// TIA Portal V15.1 export
// export: Created 2024-06-21T08:41:01.7297827Z, ExportSetting WithDefaults, DisplayName Totally Integrated Automation Portal, DisplayVersion V15.1 Update 5, DisplayName TIA Portal Openness, DisplayVersion V15.1 Update 5, DisplayName SINAMICS Startdrive Advanced, DisplayVersion V15.1, DisplayName G130, G150, S120, S150, SINAMICS MV, S210, DisplayVersion V15.1, DisplayName G110M, G120, G120C, G120D, G120P, DisplayVersion V15.1, DisplayName STEP 7 Professional, DisplayVersion V15.1 Update 5, DisplayName STEP 7 Safety, DisplayVersion V15.1, DisplayName WinCC Professional, DisplayVersion V15.1 Update 5, DisplayName SIMATIC Visualization Architect, DisplayVersion V15.1
FUNCTION_BLOCK "LCounter1Week"   // FB1801, FBD
TITLE = LCounter1Week
{ S7_Optimized_Access := 'FALSE' }
AUTHOR : VCC
FAMILY : Supervis
NAME : LCpt1W
VERSION : 1.0
// ==============================================================================
// Module create to count body produced during all shifts of the week.
// One counter per shift (moring - evening & night) per day (from monday to sunday)
// all total are foreseen.
// 
// --------------------------------------------------------------------
// Day          ! Morning shift ! Evening shift ! Night shift ! total !
// -------------!---------------!---------------!-------------!-------!
// Monday (1)   !               !               !             !       !
// -------------!---------------!---------------!-------------!-------!
// Tuesday (2)  !               !               !             !       !
// -------------!---------------!---------------!-------------!-------!
// Wednesday (3)!               !               !             !       !
// -------------!---------------!---------------!-------------!-------!
// Thursday (4) !               !               !             !       !
// -------------!---------------!---------------!-------------!-------!
// Friday (5)   !               !               !             !       !
// -------------!---------------!---------------!-------------!-------!
// Saturday (6) !               !               !             !       !
// -------------!---------------!---------------!-------------!-------!
// Sunday (7)   !               !               !             !       !
// ====================================================================
// Amount       !               !               !             !       !
// ====================================================================
// Tatal        !=============================================!       !
// ====================================================================
// 
// ==============================================================================
// stored: AutoNumber false, IsIECCheckEnabled false, SetENOAutomatically False, UDAEnableTagReadback false
   VAR_INPUT
      I_CountedInput { ExternalAccessible := 'False'; ExternalVisible := 'False'; ExternalWritable := 'False'} : Bool;   // Value to be counted
      I_MorningShift { ExternalAccessible := 'False'; ExternalVisible := 'False'; ExternalWritable := 'False'} : Bool;   // Morning shift
      I_EveningShift { ExternalAccessible := 'False'; ExternalVisible := 'False'; ExternalWritable := 'False'} : Bool;   // Evening shift
      I_NightShift { ExternalAccessible := 'False'; ExternalVisible := 'False'; ExternalWritable := 'False'} : Bool;   // NightShift
   END_VAR
   VAR_OUTPUT
      H_IAnim { ExternalAccessible := 'False'; ExternalVisible := 'False'; ExternalWritable := 'False'} : Word;   // HMI Animation of the icon
   END_VAR
   VAR DB_SPECIFIC
      H_Out : Struct   // HMI
         Anim : Word;   // HMI Animation of the object
         MorningDay1Value : Int;   // Total Production value Monday (day 1) - Morning Shift
         EveningDay1Value : Int;   // Total Production value Monday (day 1) - Evening Shift
         NightDay1Value : Int;   // Total Production value Monday (day 1) - Night Shift
         MorningDay2Value : Int;   // Total Production value Tuesday (day 2) - Morning Shift
         EveningDay2Value : Int;   // Total Production value Tuesday (day 2) - Evening Shift
         NightDay2Value : Int;   // Total Production value Tuesday (day 2) - Night Shift
         MorningDay3Value : Int;   // Total Production value Wednesday (day 3) - Morning Shift
         EveningDay3Value : Int;   // Total Production value Wednesday (day 3) - Evening Shift
         NightDay3Value : Int;   // Total Production value Wednesday (day 3) - Night Shift
         MorningDay4Value : Int;   // Total Production value Thursday (day 4) - Morning Shift
         EveningDay4Value : Int;   // Total Production value Thursday (day 4) - Evening Shift
         NightDay4Value : Int;   // Total Production value Thursday (day 4) - Night Shift
         MorningDay5Value : Int;   // Total Production value Friday (day 5) - Morning Shift
         EveningDay5Value : Int;   // Total Production value Friday (day 5) - Evening Shift
         NightDay5Value : Int;   // Total Production value Friday (day 5) - Night Shift
         MorningDay6Value : Int;   // Total Production value Saturday (day 6) - Morning Shift
         EveningDay6Value : Int;   // Total Production value Saturday (day 6) - Evening Shift
         NightDay6Value : Int;   // Total Production value Saturday (day 6) - Night Shift
         MorningDay7Value : Int;   // Production value Sunday (day 7) - Morning Shift
         EveningDay7Value : Int;   // Production value Sunday (day 7) - Evening Shift
         NightDay7Value : Int;   // Production value Sunday (day 7) - Night Shift
         Day1Value : Int;   // Total Production value Monday (day 1)
         Day2Value : Int;   // Total Production value tuesday (day 2)
         Day3Value : Int;   // Total Production value Wednesday (day 3)
         Day4Value : Int;   // Total Production value Thursday (day 4)
         Day5Value : Int;   // Total Production value Friday (day 5)
         Day6Value : Int;   // Total Production value Saturday (day 6)
         Day7Value : Int;   // Total Production value Sunday (day 7)
         TotalMorning : Int;   // Total Production value Morning
         TotalEvening : Int;   // Total Production value Evening
         TotalNight : Int;   // Total Production value Night
         WeekValue : Int;   // Total Production value Week
         TotalValue : DInt;   // Total production value
         DBnr : Int;   // HMI Animation DB number
      END_STRUCT;
      CountedInputPulse { ExternalAccessible := 'False'; ExternalVisible := 'False'; ExternalWritable := 'False'} : Bool;   // Pulse of value to be counted
      CountUp { ExternalAccessible := 'False'; ExternalVisible := 'False'; ExternalWritable := 'False'} : Bool;   // Pulse of value to be counted
      MorningShiftPulse { ExternalAccessible := 'False'; ExternalVisible := 'False'; ExternalWritable := 'False'} : Bool;   // Pulse of Morning shift
      MorningPulse { ExternalAccessible := 'False'; ExternalVisible := 'False'; ExternalWritable := 'False'} : Bool;   // Pulse of Morning shift
      Day1 { ExternalAccessible := 'False'; ExternalVisible := 'False'; ExternalWritable := 'False'} : Bool;   // Day 1 = Monday
      Day2 { ExternalAccessible := 'False'; ExternalVisible := 'False'; ExternalWritable := 'False'} : Bool;   // Day 2 = Tuesday
      Day3 { ExternalAccessible := 'False'; ExternalVisible := 'False'; ExternalWritable := 'False'} : Bool;   // Day 3 = Wednesday
      Day4 { ExternalAccessible := 'False'; ExternalVisible := 'False'; ExternalWritable := 'False'} : Bool;   // Day 4 = Thursday
      Day5 { ExternalAccessible := 'False'; ExternalVisible := 'False'; ExternalWritable := 'False'} : Bool;   // Day 5 = Friday
      Day6 { ExternalAccessible := 'False'; ExternalVisible := 'False'; ExternalWritable := 'False'} : Bool;   // Day 6 = Saturday
      Day7 { ExternalAccessible := 'False'; ExternalVisible := 'False'; ExternalWritable := 'False'} : Bool;   // Day 7 = Sunday
      MorningValue { ExternalAccessible := 'False'; ExternalVisible := 'False'; ExternalWritable := 'False'} : Int;   // Morning production value
      EveningValue { ExternalAccessible := 'False'; ExternalVisible := 'False'; ExternalWritable := 'False'} : Int;   // Evening production value
      NightValue { ExternalAccessible := 'False'; ExternalVisible := 'False'; ExternalWritable := 'False'} : Int;   // Night production value
      MorningDay1Value { ExternalAccessible := 'False'; ExternalVisible := 'False'; ExternalWritable := 'False'} : Int;   // Total Production value Monday (day 1) - Morning Shift
      EveningDay1Value { ExternalAccessible := 'False'; ExternalVisible := 'False'; ExternalWritable := 'False'} : Int;   // Total Production value Monday (day 1) - Evening Shift
      NightDay1Value { ExternalAccessible := 'False'; ExternalVisible := 'False'; ExternalWritable := 'False'} : Int;   // Total Production value Monday (day 1) - Night Shift
      MorningDay2Value { ExternalAccessible := 'False'; ExternalVisible := 'False'; ExternalWritable := 'False'} : Int;   // Total Production value Tuesday (day 2) - Morning Shift
      EveningDay2Value { ExternalAccessible := 'False'; ExternalVisible := 'False'; ExternalWritable := 'False'} : Int;   // Total Production value Tuesday (day 2) - Evening Shift
      NightDay2Value { ExternalAccessible := 'False'; ExternalVisible := 'False'; ExternalWritable := 'False'} : Int;   // Total Production value Tuesday (day 2) - Night Shift
      MorningDay3Value { ExternalAccessible := 'False'; ExternalVisible := 'False'; ExternalWritable := 'False'} : Int;   // Total Production value Wednesday (day 3) - Morning Shift
      EveningDay3Value { ExternalAccessible := 'False'; ExternalVisible := 'False'; ExternalWritable := 'False'} : Int;   // Total Production value Wednesday (day 3) - Evening Shift
      NightDay3Value { ExternalAccessible := 'False'; ExternalVisible := 'False'; ExternalWritable := 'False'} : Int;   // Total Production value Wednesday (day 3) - Night Shift
      MorningDay4Value { ExternalAccessible := 'False'; ExternalVisible := 'False'; ExternalWritable := 'False'} : Int;   // Total Production value Thursday (day 4) - Morning Shift
      EveningDay4Value { ExternalAccessible := 'False'; ExternalVisible := 'False'; ExternalWritable := 'False'} : Int;   // Total Production value Thursday (day 4) - Evening Shift
      NightDay4Value { ExternalAccessible := 'False'; ExternalVisible := 'False'; ExternalWritable := 'False'} : Int;   // Total Production value Thursday (day 4) - Night Shift
      MorningDay5Value { ExternalAccessible := 'False'; ExternalVisible := 'False'; ExternalWritable := 'False'} : Int;   // Total Production value Friday (day 5) - Morning Shift
      EveningDay5Value { ExternalAccessible := 'False'; ExternalVisible := 'False'; ExternalWritable := 'False'} : Int;   // Total Production value Friday (day 5) - Evening Shift
      NightDay5Value { ExternalAccessible := 'False'; ExternalVisible := 'False'; ExternalWritable := 'False'} : Int;   // Total Production value Friday (day 5) - Night Shift
      MorningDay6Value { ExternalAccessible := 'False'; ExternalVisible := 'False'; ExternalWritable := 'False'} : Int;   // Total Production value Saturday (day 6) - Morning Shift
      EveningDay6Value { ExternalAccessible := 'False'; ExternalVisible := 'False'; ExternalWritable := 'False'} : Int;   // Total Production value Saturday (day 6) - Evening Shift
      NightDay6Value { ExternalAccessible := 'False'; ExternalVisible := 'False'; ExternalWritable := 'False'} : Int;   // Total Production value Saturday (day 6) - Night Shift
      MorningDay7Value { ExternalAccessible := 'False'; ExternalVisible := 'False'; ExternalWritable := 'False'} : Int;   // Production value Sunday (day 7) - Morning Shift
      EveningDay7Value { ExternalAccessible := 'False'; ExternalVisible := 'False'; ExternalWritable := 'False'} : Int;   // Production value Sunday (day 7) - Evening Shift
      NightDay7Value { ExternalAccessible := 'False'; ExternalVisible := 'False'; ExternalWritable := 'False'} : Int;   // Production value Sunday (day 7) - Night Shift
      Day1Value { ExternalAccessible := 'False'; ExternalVisible := 'False'; ExternalWritable := 'False'} : Int;   // Total Production value Monday (day 1)
      Day2Value { ExternalAccessible := 'False'; ExternalVisible := 'False'; ExternalWritable := 'False'} : Int;   // Total Production value tuesday (day 2)
      Day3Value { ExternalAccessible := 'False'; ExternalVisible := 'False'; ExternalWritable := 'False'} : Int;   // Total Production value Wednesday (day 3)
      Day4Value { ExternalAccessible := 'False'; ExternalVisible := 'False'; ExternalWritable := 'False'} : Int;   // Total Production value Thursday (day 4)
      Day5Value { ExternalAccessible := 'False'; ExternalVisible := 'False'; ExternalWritable := 'False'} : Int;   // Total Production value Friday (day 5)
      Day6Value { ExternalAccessible := 'False'; ExternalVisible := 'False'; ExternalWritable := 'False'} : Int;   // Total Production value Saturday (day 6)
      Day7Value { ExternalAccessible := 'False'; ExternalVisible := 'False'; ExternalWritable := 'False'} : Int;   // Total Production value Sunday (day 7)
      WeekValue { ExternalAccessible := 'False'; ExternalVisible := 'False'; ExternalWritable := 'False'} : Int;   // Total Production value Week
      TotalValue { ExternalAccessible := 'False'; ExternalVisible := 'False'; ExternalWritable := 'False'} : DInt;   // Total production value
      DBnr { ExternalAccessible := 'False'; ExternalVisible := 'False'; ExternalWritable := 'False'} : Int;   // HMI DB number
   END_VAR
   VAR_TEMP   // added for the SCL form of the ladder/FBD networks
      _w1 : Bool;
   END_VAR
BEGIN

NETWORK
TITLE = **** 1 - Inputs **** DB number
// DB number
      L     DINO;
      T     #DBnr;

REGION Network 2: **** 4.4 - Machine status - Calculated **** Total production counter
   // Total production counter
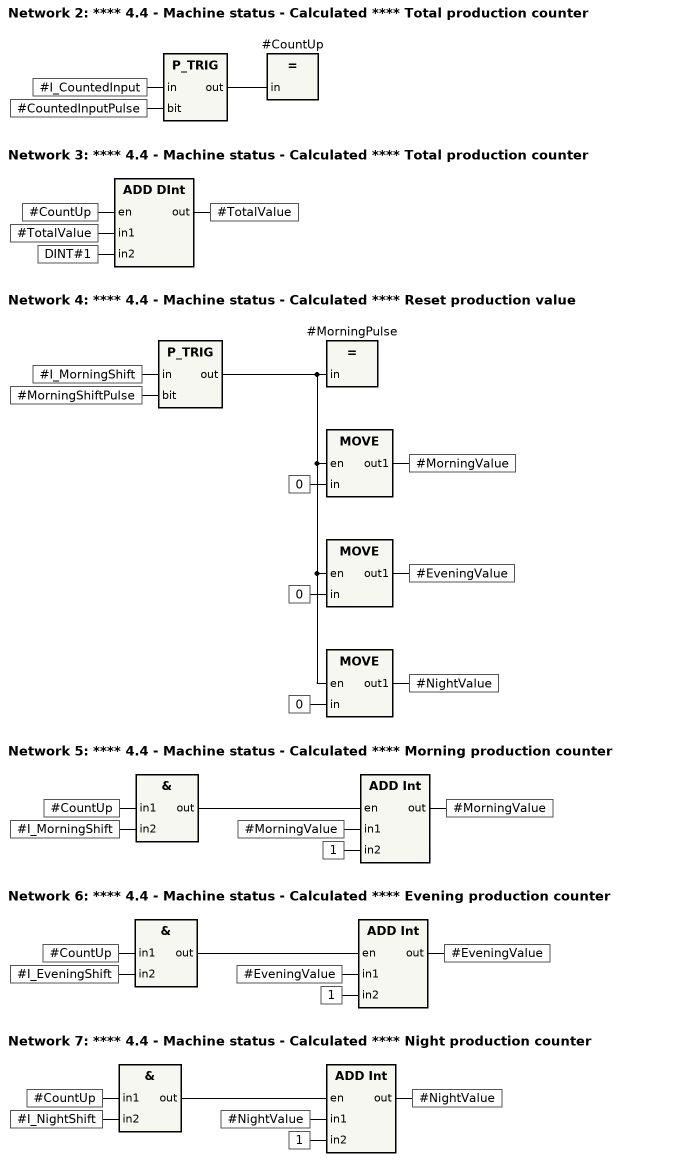
   #_w1 := #I_CountedInput AND NOT #CountedInputPulse;   // rising edge
   #CountedInputPulse := #I_CountedInput;
   #CountUp := #_w1;
END_REGION

REGION Network 3: **** 4.4 - Machine status - Calculated **** Total production counter
   // Total production counter
   IF #CountUp THEN #TotalValue := #TotalValue + DINT#1; END_IF;
END_REGION

REGION Network 4: **** 4.4 - Machine status - Calculated **** Reset production value
   // Reset production value
   #_w1 := #I_MorningShift AND NOT #MorningShiftPulse;   // rising edge
   #MorningShiftPulse := #I_MorningShift;
   #MorningPulse := #_w1;
   IF #_w1 THEN
       #MorningValue := 0;
       #EveningValue := 0;
       #NightValue := 0;
   END_IF;
END_REGION

REGION Network 5: **** 4.4 - Machine status - Calculated **** Morning production counter
   // Morning production counter
   IF #CountUp AND #I_MorningShift THEN #MorningValue := #MorningValue + 1; END_IF;
END_REGION

REGION Network 6: **** 4.4 - Machine status - Calculated **** Evening production counter
   // Evening production counter
   IF #CountUp AND #I_EveningShift THEN #EveningValue := #EveningValue + 1; END_IF;
END_REGION

REGION Network 7: **** 4.4 - Machine status - Calculated **** Night production counter
   // Night production counter
   IF #CountUp AND #I_NightShift THEN #NightValue := #NightValue + 1; END_IF;
END_REGION

REGION Network 8: **** 4.4 - Machine status - Calculated **** Set Monday - reset other days
   // Set Monday - reset other days
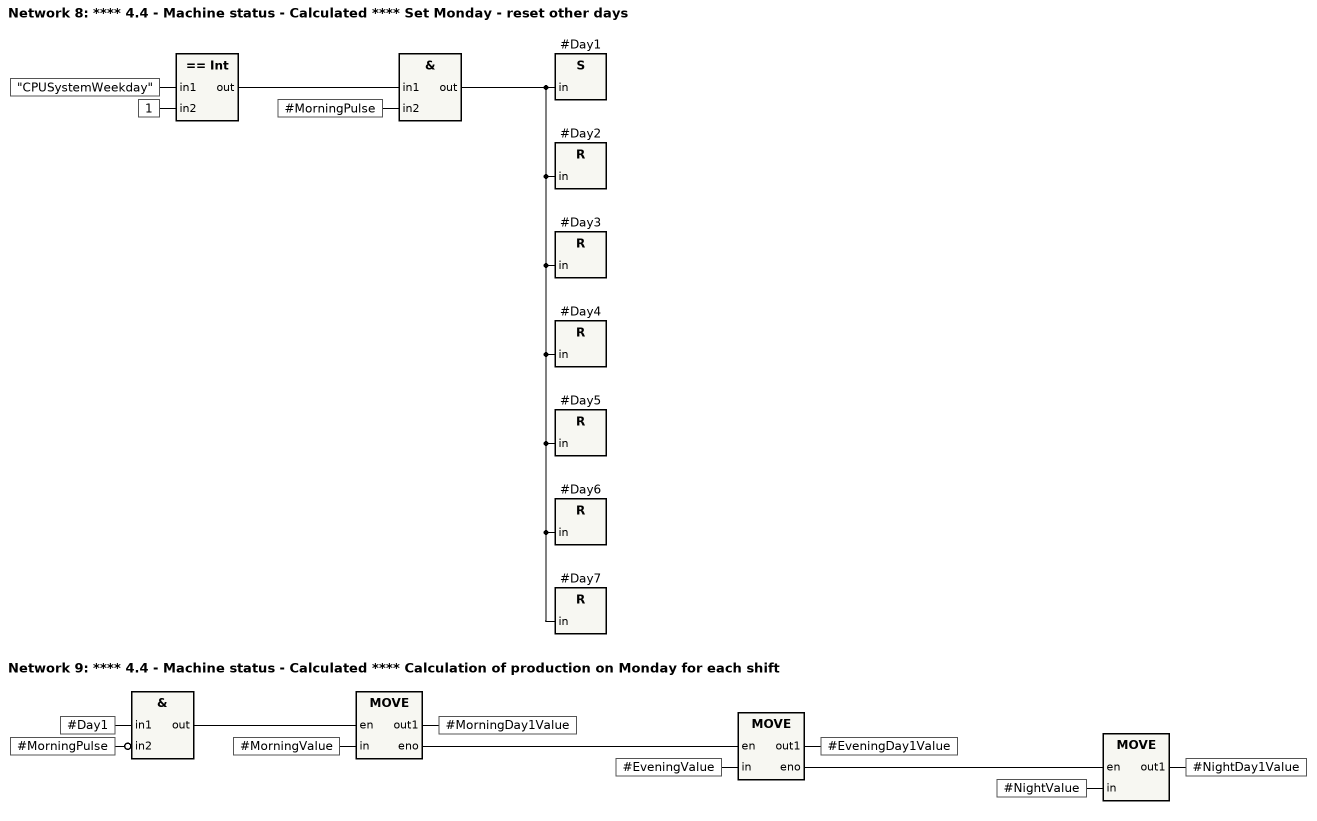
   IF ("CPUSystemWeekday" = 1) AND #MorningPulse THEN
       #Day1 := TRUE;
       #Day2 := FALSE;
       #Day3 := FALSE;
       #Day4 := FALSE;
       #Day5 := FALSE;
       #Day6 := FALSE;
       #Day7 := FALSE;
   END_IF;
END_REGION

REGION Network 9: **** 4.4 - Machine status - Calculated **** Calculation of production on Monday for each shift
   // Calculation of production on Monday for each shift
   // ENO of a box is taken as its EN; it also drops when the box reports an error
   IF #Day1 AND NOT #MorningPulse THEN
       #MorningDay1Value := #MorningValue;
       #EveningDay1Value := #EveningValue;
       #NightDay1Value := #NightValue;
   END_IF;
END_REGION

NETWORK
TITLE = **** 4.4 - Machine status - Calculated **** Total production on Monday
// Total production on Monday
      L     #MorningDay1Value;  // amount of bodies on day 1 - Morning shift (Monday)
      L     #EveningDay1Value;  // amount of bodies on day 1 - Evening shift (Monday)
      +I;
      L     #NightDay1Value;  // amount of bodies on day 1 - Night shift (Monday)
      +I;
      T     #Day1Value;  // amount of bodies on day 1 (Monday)

REGION Network 11: **** 4.4 - Machine status - Calculated **** Set Tuesday - reset other days
   // Set Tuesday - reset other days
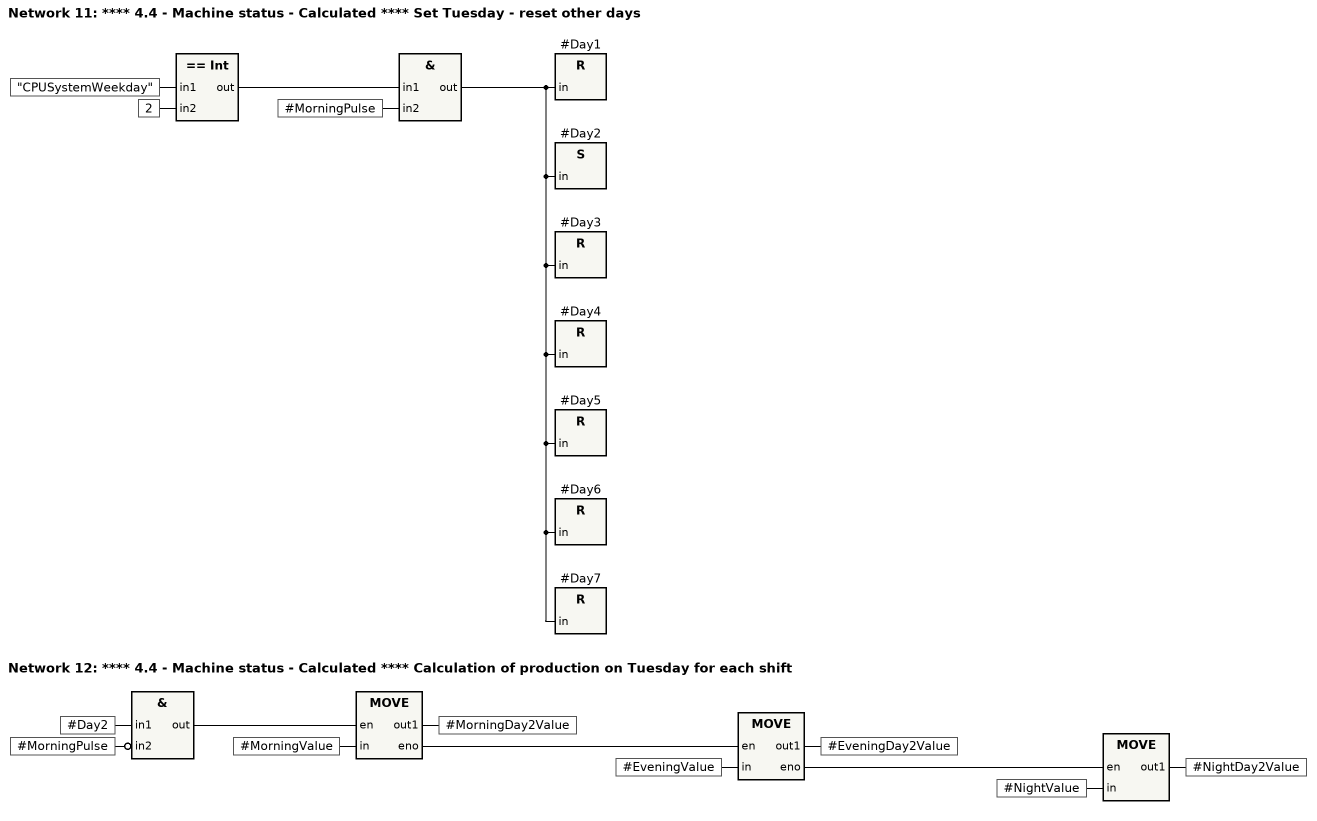
   IF ("CPUSystemWeekday" = 2) AND #MorningPulse THEN
       #Day1 := FALSE;
       #Day2 := TRUE;
       #Day3 := FALSE;
       #Day4 := FALSE;
       #Day5 := FALSE;
       #Day6 := FALSE;
       #Day7 := FALSE;
   END_IF;
END_REGION

REGION Network 12: **** 4.4 - Machine status - Calculated **** Calculation of production on Tuesday for each shift
   // Calculation of production on Tuesday for each shift
   // ENO of a box is taken as its EN; it also drops when the box reports an error
   IF #Day2 AND NOT #MorningPulse THEN
       #MorningDay2Value := #MorningValue;
       #EveningDay2Value := #EveningValue;
       #NightDay2Value := #NightValue;
   END_IF;
END_REGION

NETWORK
TITLE = **** 4.4 - Machine status - Calculated **** Total production on Thuesday
// Total production on Thuesday
      L     #MorningDay2Value;  // amount of bodies on day 2 - Morning shift (Tuesday)
      L     #EveningDay2Value;  // amount of bodies on day 2 - Evening shift (Tuesday)
      +I;
      L     #NightDay2Value;  // amount of bodies on day 2 - Night shift (Tuesday)
      +I;
      T     #Day2Value;  // amount of bodies on day 2 (Tuesday)

REGION Network 14: **** 4.4 - Machine status - Calculated **** Set Wednesday - reset other days
   // Set Wednesday - reset other days
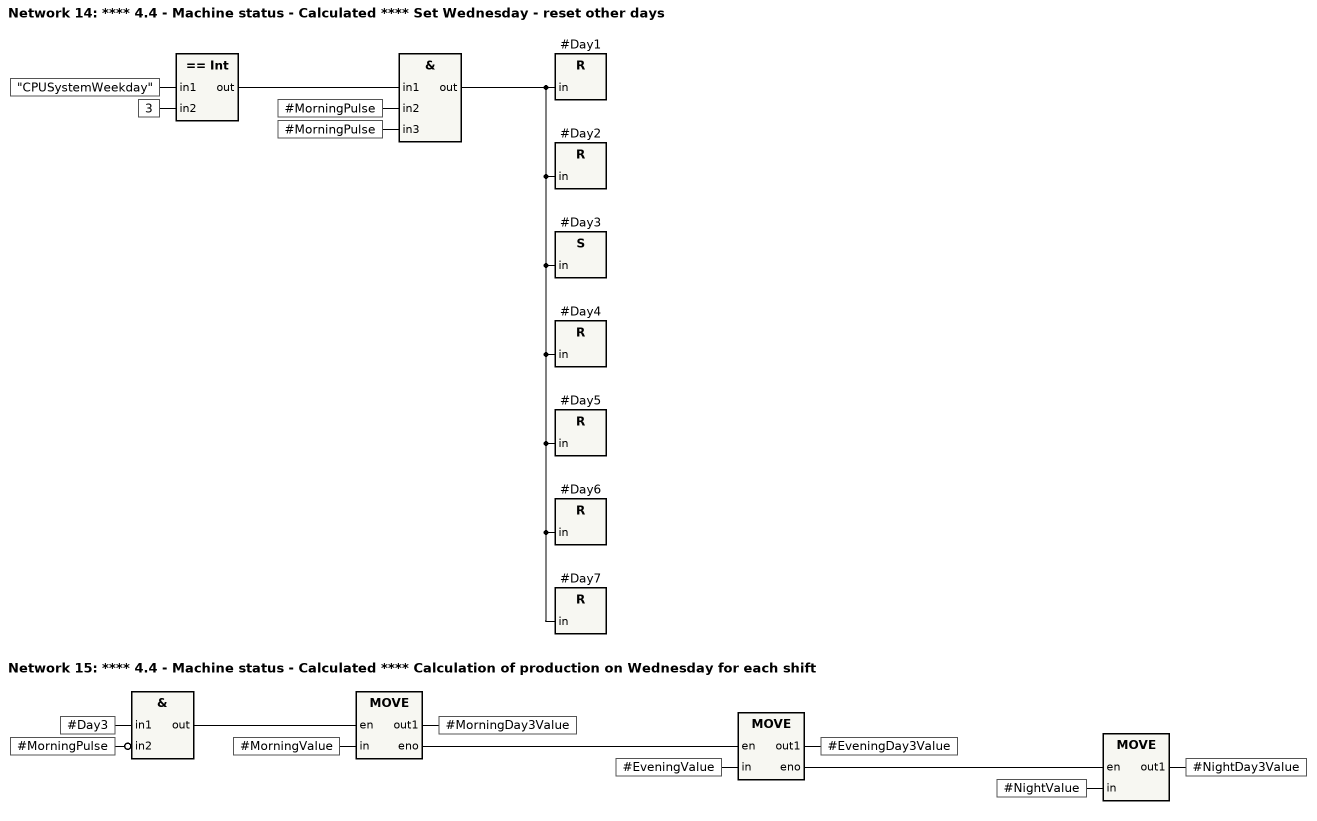
   IF ("CPUSystemWeekday" = 3) AND #MorningPulse AND #MorningPulse THEN
       #Day1 := FALSE;
       #Day2 := FALSE;
       #Day3 := TRUE;
       #Day4 := FALSE;
       #Day5 := FALSE;
       #Day6 := FALSE;
       #Day7 := FALSE;
   END_IF;
END_REGION

REGION Network 15: **** 4.4 - Machine status - Calculated **** Calculation of production on Wednesday for each shift
   // Calculation of production on Wednesday for each shift
   // ENO of a box is taken as its EN; it also drops when the box reports an error
   IF #Day3 AND NOT #MorningPulse THEN
       #MorningDay3Value := #MorningValue;
       #EveningDay3Value := #EveningValue;
       #NightDay3Value := #NightValue;
   END_IF;
END_REGION

NETWORK
TITLE = **** 4.4 - Machine status - Calculated **** Total production on Wednesday
// Total production on Wednesday
      L     #MorningDay3Value;  // amount of bodies on day 3 - Morning shift (Wednesday)
      L     #EveningDay3Value;  // amount of bodies on day 3 - Evening shift (Wednesday)
      +I;
      L     #NightDay3Value;  // amount of bodies on day 3 - Night shift (Wednesday)
      +I;
      T     #Day3Value;  // amount of bodies on day 3 (Wednesday)

REGION Network 17: **** 4.4 - Machine status - Calculated **** Set Thursday - reset other days
   // Set Thursday - reset other days
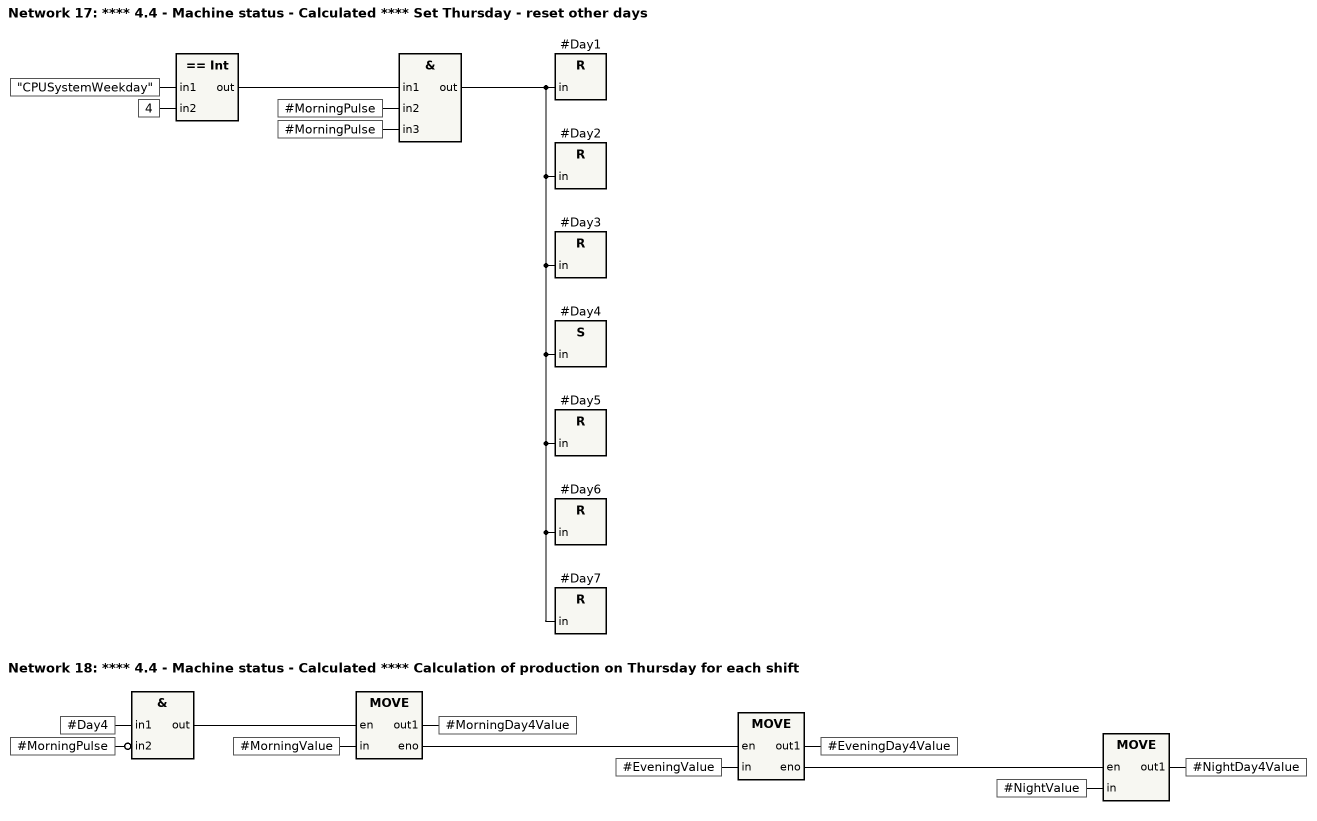
   IF ("CPUSystemWeekday" = 4) AND #MorningPulse AND #MorningPulse THEN
       #Day1 := FALSE;
       #Day2 := FALSE;
       #Day3 := FALSE;
       #Day4 := TRUE;
       #Day5 := FALSE;
       #Day6 := FALSE;
       #Day7 := FALSE;
   END_IF;
END_REGION

REGION Network 18: **** 4.4 - Machine status - Calculated **** Calculation of production on Thursday for each shift
   // Calculation of production on Thursday for each shift
   // ENO of a box is taken as its EN; it also drops when the box reports an error
   IF #Day4 AND NOT #MorningPulse THEN
       #MorningDay4Value := #MorningValue;
       #EveningDay4Value := #EveningValue;
       #NightDay4Value := #NightValue;
   END_IF;
END_REGION

NETWORK
TITLE = **** 4.4 - Machine status - Calculated **** Total production on Thursday
// Total production on Thursday
      L     #MorningDay4Value;  // amount of bodies on day 4 - Morning shift (Thursday)
      L     #EveningDay4Value;  // amount of bodies on day 4 - Evening shift (Thursday)
      +I;
      L     #NightDay4Value;  // amount of bodies on day 4 - Night shift (Thursday)
      +I;
      T     #Day4Value;  // amount of bodies on day 4 (Thursday)

REGION Network 20: **** 4.4 - Machine status - Calculated **** Set Friday - reset other days
   // Set Friday - reset other days
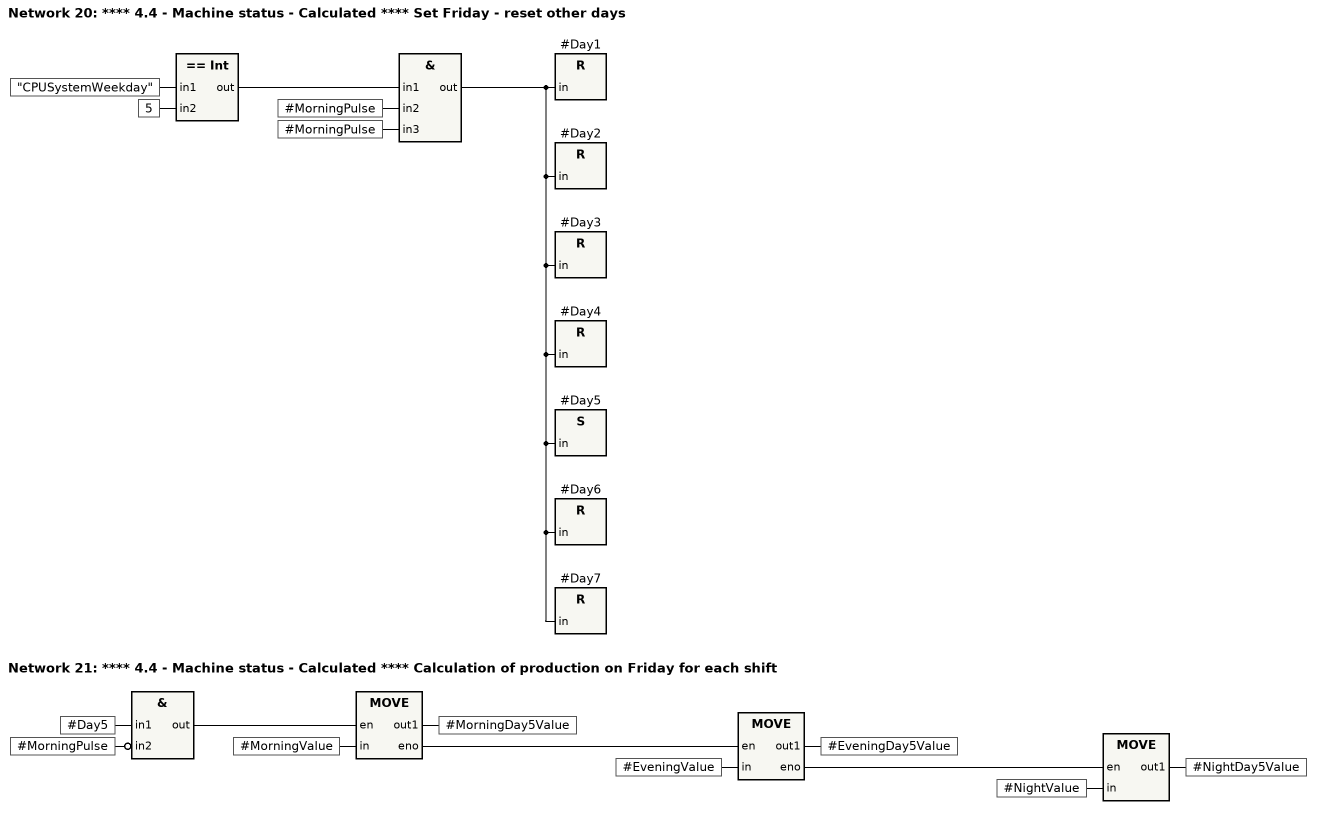
   IF ("CPUSystemWeekday" = 5) AND #MorningPulse AND #MorningPulse THEN
       #Day1 := FALSE;
       #Day2 := FALSE;
       #Day3 := FALSE;
       #Day4 := FALSE;
       #Day5 := TRUE;
       #Day6 := FALSE;
       #Day7 := FALSE;
   END_IF;
END_REGION

REGION Network 21: **** 4.4 - Machine status - Calculated **** Calculation of production on Friday for each shift
   // Calculation of production on Friday for each shift
   // ENO of a box is taken as its EN; it also drops when the box reports an error
   IF #Day5 AND NOT #MorningPulse THEN
       #MorningDay5Value := #MorningValue;
       #EveningDay5Value := #EveningValue;
       #NightDay5Value := #NightValue;
   END_IF;
END_REGION

NETWORK
TITLE = **** 4.4 - Machine status - Calculated **** total production on Friday
// total production on Friday
      L     #MorningDay5Value;  // amount of bodies on day 5 - Morning shift (Friday)
      L     #EveningDay5Value;  // amount of bodies on day 5 - Evening shift (Friday)
      +I;
      L     #NightDay5Value;  // amount of bodies on day 5 - Night shift (Friday)
      +I;
      T     #Day5Value;  // amount of bodies on day 5 (Friday)

REGION Network 23: **** 4.4 - Machine status - Calculated **** Set Saturday - Reset other days
   // Set Saturday - Reset other days
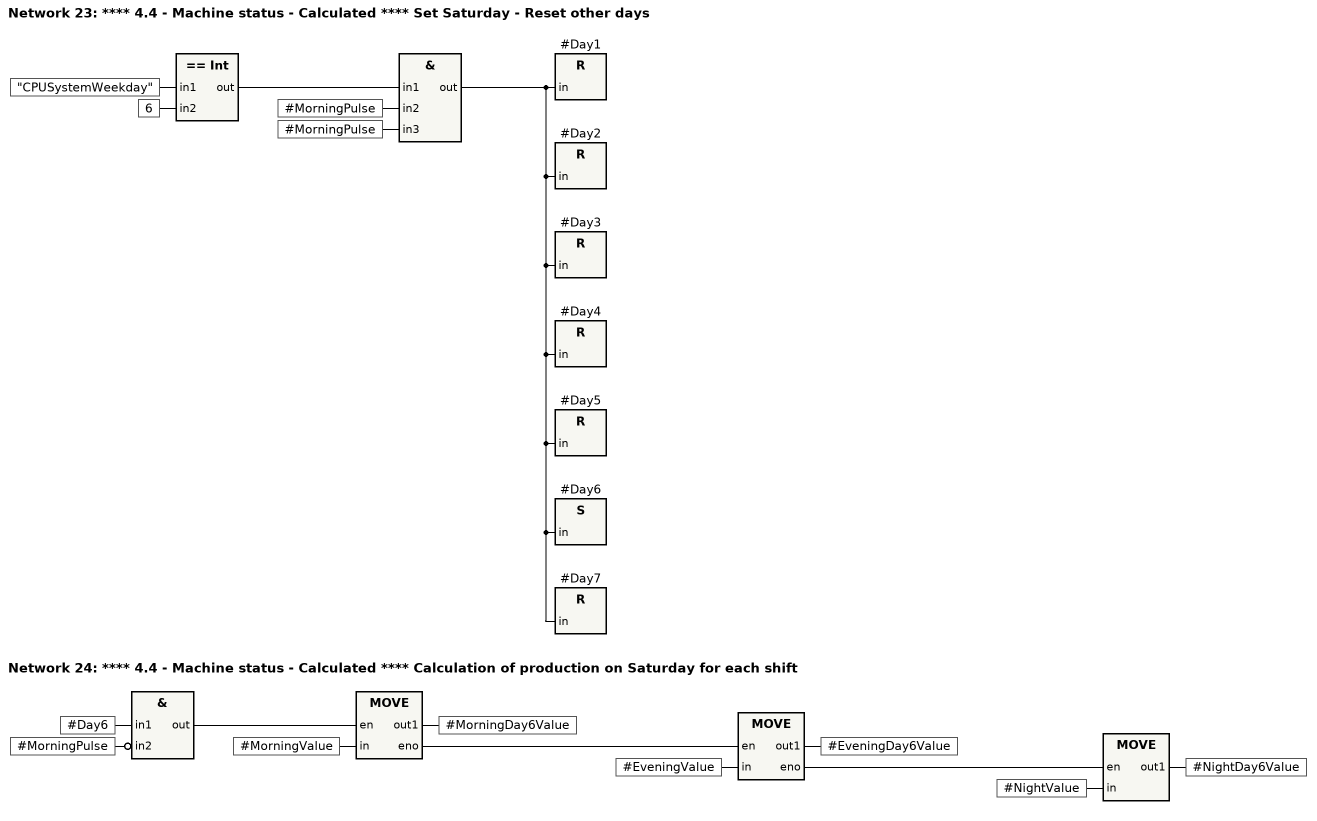
   IF ("CPUSystemWeekday" = 6) AND #MorningPulse AND #MorningPulse THEN
       #Day1 := FALSE;
       #Day2 := FALSE;
       #Day3 := FALSE;
       #Day4 := FALSE;
       #Day5 := FALSE;
       #Day6 := TRUE;
       #Day7 := FALSE;
   END_IF;
END_REGION

REGION Network 24: **** 4.4 - Machine status - Calculated **** Calculation of production on Saturday for each shift
   // Calculation of production on Saturday for each shift
   // ENO of a box is taken as its EN; it also drops when the box reports an error
   IF #Day6 AND NOT #MorningPulse THEN
       #MorningDay6Value := #MorningValue;
       #EveningDay6Value := #EveningValue;
       #NightDay6Value := #NightValue;
   END_IF;
END_REGION

NETWORK
TITLE = **** 4.4 - Machine status - Calculated **** total production on Saturday
// total production on Saturday
      L     #MorningDay6Value;  // amount of bodies on day 6 - Morning shift (Saturday)
      L     #EveningDay6Value;  // amount of bodies on day 6 - Evening shift (Saturday)
      +I;
      L     #NightDay6Value;  // amount of bodies on day 6 - Night shift (Saturday)
      +I;
      T     #Day6Value;  // amount of bodies on day 6 (Saturday)

REGION Network 26: **** 4.4 - Machine status - Calculated **** Set Sunday - Reset other days
   // Set Sunday - Reset other days
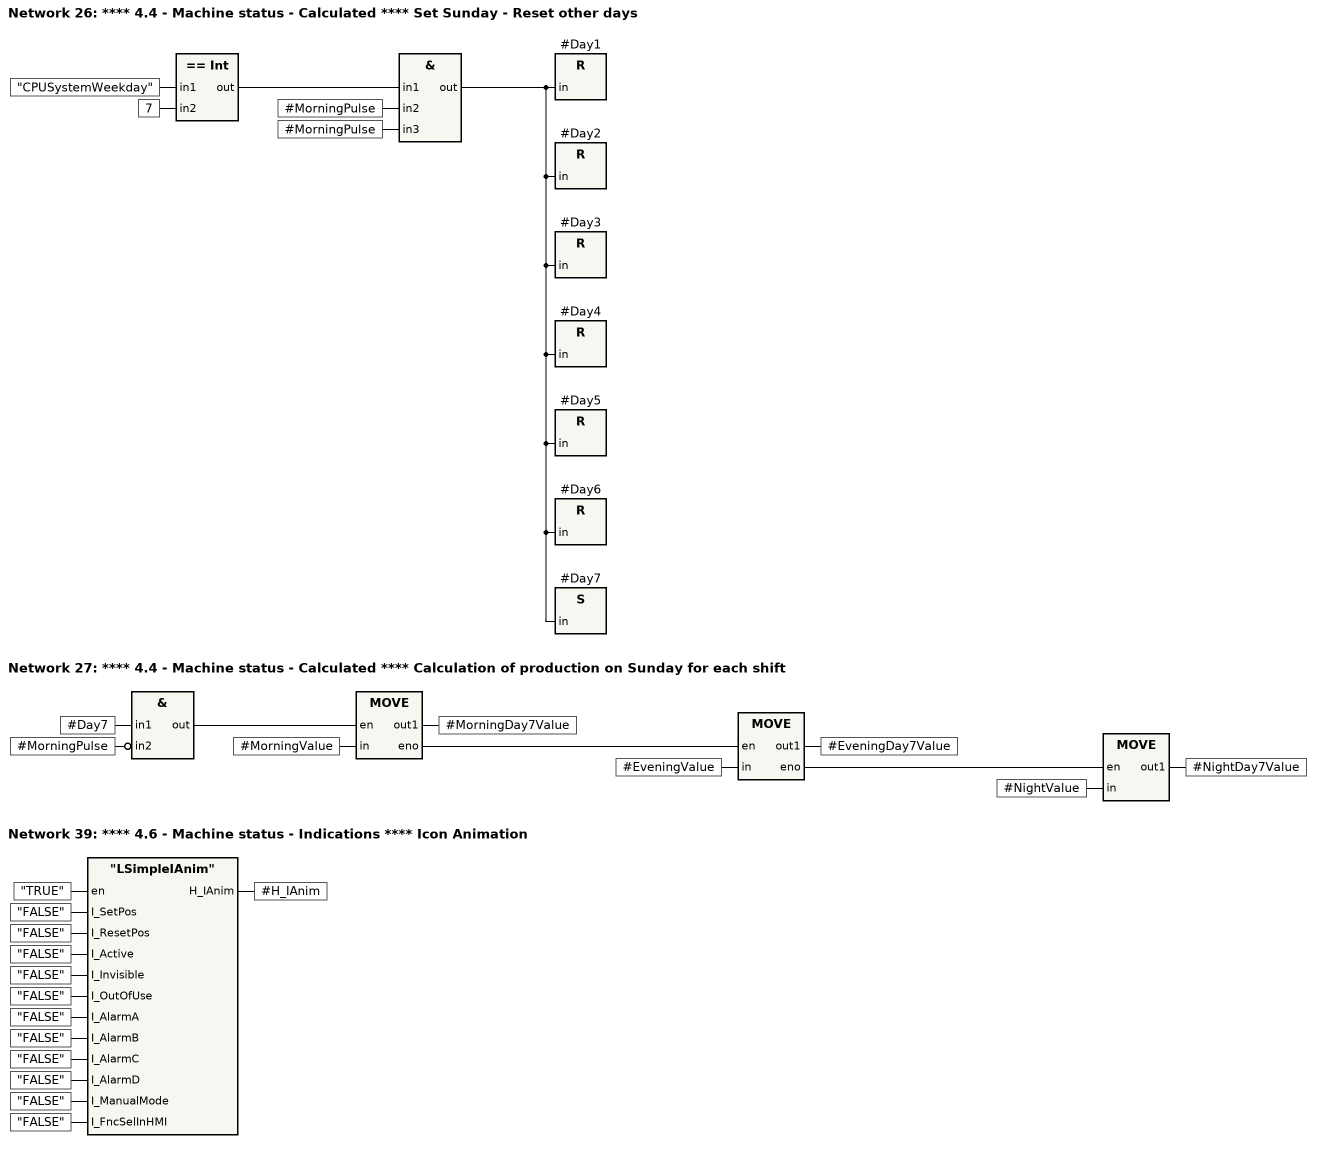
   IF ("CPUSystemWeekday" = 7) AND #MorningPulse AND #MorningPulse THEN
       #Day1 := FALSE;
       #Day2 := FALSE;
       #Day3 := FALSE;
       #Day4 := FALSE;
       #Day5 := FALSE;
       #Day6 := FALSE;
       #Day7 := TRUE;
   END_IF;
END_REGION

REGION Network 27: **** 4.4 - Machine status - Calculated **** Calculation of production on Sunday for each shift
   // Calculation of production on Sunday for each shift
   // ENO of a box is taken as its EN; it also drops when the box reports an error
   IF #Day7 AND NOT #MorningPulse THEN
       #MorningDay7Value := #MorningValue;
       #EveningDay7Value := #EveningValue;
       #NightDay7Value := #NightValue;
   END_IF;
END_REGION

NETWORK
TITLE = **** 4.4 - Machine status - Calculated **** Total production on Sunday
// Total production on Sunday
      L     #MorningDay7Value;  // amount of bodies on day 7 - Morning shift (Sunday)
      L     #EveningDay7Value;  // amount of bodies on day 7 - Evening shift (Sunday)
      +I;
      L     #NightDay7Value;  // amount of bodies on day 7 - Night shift (Sunday)
      +I;
      T     #Day7Value;  // amount of bodies on day 7 (Sunday)

NETWORK
TITLE = **** 4.4 - Machine status - Calculated **** Production value Morning shift
// Production value Morning shift
      A     #Day1;  // Day 1 (Monday)
      JNB   MD1;
      L     #MorningDay1Value;  // amount of bodies on day 1 - Morning shift (Monday)
      T     #H_Out.TotalMorning;  // copy to HMI
MD1:  NOP   0;

      A     #Day2;  // Day 2 (tuesday)
      JNB   MD2;
      L     #MorningDay1Value;  // amount of bodies on day 1 - Morning shift (Monday)
      L     #MorningDay2Value;  // amount of bodies on day 2 - Morning shift (Tuesday)
      T     #H_Out.TotalMorning;  // copy to HMI
MD2:  NOP   0;

      A     #Day3;  // Day 3 (Wednesday)
      JNB   MD3;
      L     #MorningDay1Value;  // amount of bodies on day 1 - Morning shift (Monday)
      L     #MorningDay2Value;  // amount of bodies on day 2 - Morning shift (Tuesday)
      +I;
      L     #MorningDay3Value;  // amount of bodies on day 3 - Morning shift (Wednesday)
      +I;
      T     #H_Out.TotalMorning;  // copy to HMI
MD3:  NOP   0;

      A     #Day4;  // Day 4 (tuesday)
      JNB   MD4;
      L     #MorningDay1Value;  // amount of bodies on day 1 - Morning shift (Monday)
      L     #MorningDay2Value;  // amount of bodies on day 2 - Morning shift (Tuesday)
      +I;
      L     #MorningDay3Value;  // amount of bodies on day 3 - Morning shift (Wednesday)
      +I;
      L     #MorningDay4Value;  // amount of bodies on day 4 - Morning shift (Thursday)
      +I;
      T     #H_Out.TotalMorning;  // copy to HMI
MD4:  NOP   0;

      A     #Day5;  // Day 5 (Friday)
      JNB   MD5;
      L     #MorningDay1Value;  // amount of bodies on day 1 - Morning shift (Monday)
      L     #MorningDay2Value;  // amount of bodies on day 2 - Morning shift (Tuesday)
      +I;
      L     #MorningDay3Value;  // amount of bodies on day 3 - Morning shift (Wednesday)
      +I;
      L     #MorningDay4Value;  // amount of bodies on day 4 - Morning shift (Thursday)
      +I;
      L     #MorningDay5Value;  // amount of bodies on day 5 - Morning shift (Friday)
      +I;
      T     #H_Out.TotalMorning;  // copy to HMI
MD5:  NOP   0;

      A     #Day6;  // Day 6 (Saturday)
      JNB   MD6;
      L     #MorningDay1Value;  // amount of bodies on day 1 - Morning shift (Monday)
      L     #MorningDay2Value;  // amount of bodies on day 2 - Morning shift (Tuesday)
      +I;
      L     #MorningDay3Value;  // amount of bodies on day 3 - Morning shift (Wednesday)
      +I;
      L     #MorningDay4Value;  // amount of bodies on day 4 - Morning shift (Thursday)
      +I;
      L     #MorningDay5Value;  // amount of bodies on day 5 - Morning shift (Friday)
      +I;
      L     #MorningDay6Value;  // amount of bodies on day 6 - Morning shift (Saturday)
      +I;
      T     #H_Out.TotalMorning;  // copy to HMI
MD6:  NOP   0;

      A     #Day7;  // Day 7 (Sunday)
      JNB   MD7;
      L     #MorningDay1Value;  // amount of bodies on day 1 - Morning shift (Monday)
      L     #MorningDay2Value;  // amount of bodies on day 2 - Morning shift (Tuesday)
      +I;
      L     #MorningDay3Value;  // amount of bodies on day 3 - Morning shift (Wednesday)
      +I;
      L     #MorningDay4Value;  // amount of bodies on day 4 - Morning shift (Thursday)
      +I;
      L     #MorningDay5Value;  // amount of bodies on day 5 - Morning shift (Friday)
      +I;
      L     #MorningDay6Value;  // amount of bodies on day 6 - Morning shift (Saturday)
      +I;
      L     #MorningDay7Value;  // amount of bodies on day 7 - Morning shift (Sunday)
      +I;
      T     #H_Out.TotalMorning;  // copy to HMI
MD7:  NOP   0;


NETWORK
TITLE = **** 4.4 - Machine status - Calculated **** Production value Evening shift
// Production value Evening shift
      A     #Day1;  // Day 1 (Monday)
      JNB   ED1;
      L     #EveningDay1Value;  // amount of bodies on day 1 - Evening shift (Monday)
      T     #H_Out.TotalEvening;  // copy to HMI
ED1:  NOP   0;

      A     #Day2;  // Day 2 (tuesday)
      JNB   ED2;
      L     #EveningDay1Value;  // amount of bodies on day 1 - Evening shift (Monday)
      L     #EveningDay2Value;  // amount of bodies on day 2 - Evening shift (Tuesday)
      T     #H_Out.TotalEvening;  // copy to HMI
ED2:  NOP   0;

      A     #Day3;  // Day 3 (Wednesday)
      JNB   ED3;
      L     #EveningDay1Value;  // amount of bodies on day 1 - Evening shift (Monday)
      L     #EveningDay2Value;  // amount of bodies on day 2 - Evening shift (Tuesday)
      +I;
      L     #EveningDay3Value;  // amount of bodies on day 3 - Evening shift (Wednesday)
      +I;
      T     #H_Out.TotalEvening;  // copy to HMI
ED3:  NOP   0;

      A     #Day4;  // Day 4 (tuesday)
      JNB   ED4;
      L     #EveningDay1Value;  // amount of bodies on day 1 - Evening shift (Monday)
      L     #EveningDay2Value;  // amount of bodies on day 2 - Evening shift (Tuesday)
      +I;
      L     #EveningDay3Value;  // amount of bodies on day 3 - Evening shift (Wednesday)
      +I;
      L     #EveningDay4Value;  // amount of bodies on day 4 - Evening shift (Thursday)
      +I;
      T     #H_Out.TotalEvening;  // copy to HMI
ED4:  NOP   0;

      A     #Day5;  // Day 5 (Friday)
      JNB   ED5;
      L     #EveningDay1Value;  // amount of bodies on day 1 - Evening shift (Monday)
      L     #EveningDay2Value;  // amount of bodies on day 2 - Evening shift (Tuesday)
      +I;
      L     #EveningDay3Value;  // amount of bodies on day 3 - Evening shift (Wednesday)
      +I;
      L     #EveningDay4Value;  // amount of bodies on day 4 - Evening shift (Thursday)
      +I;
      L     #EveningDay5Value;  // amount of bodies on day 5 - Evening shift (Friday)
      +I;
      T     #H_Out.TotalEvening;  // copy to HMI
ED5:  NOP   0;

      A     #Day6;  // Day 6 (Saturday)
      JNB   ED6;
      L     #EveningDay1Value;  // amount of bodies on day 1 - Evening shift (Monday)
      L     #EveningDay2Value;  // amount of bodies on day 2 - Evening shift (Tuesday)
      +I;
      L     #EveningDay3Value;  // amount of bodies on day 3 - Evening shift (Wednesday)
      +I;
      L     #EveningDay4Value;  // amount of bodies on day 4 - Evening shift (Thursday)
      +I;
      L     #EveningDay5Value;  // amount of bodies on day 5 - Evening shift (Friday)
      +I;
      L     #EveningDay6Value;  // amount of bodies on day 6 - Evening shift (Saturday)
      +I;
      T     #H_Out.TotalEvening;  // copy to HMI
ED6:  NOP   0;

      A     #Day7;  // Day 7 (Sunday)
      JNB   ED7;
      L     #EveningDay1Value;  // amount of bodies on day 1 - Evening shift (Monday)
      L     #EveningDay2Value;  // amount of bodies on day 2 - Evening shift (Tuesday)
      +I;
      L     #EveningDay3Value;  // amount of bodies on day 3 - Evening shift (Wednesday)
      +I;
      L     #EveningDay4Value;  // amount of bodies on day 4 - Evening shift (Thursday)
      +I;
      L     #EveningDay5Value;  // amount of bodies on day 5 - Evening shift (Friday)
      +I;
      L     #EveningDay6Value;  // amount of bodies on day 6 - Evening shift (Saturday)
      +I;
      L     #EveningDay7Value;  // amount of bodies on day 7 - Evening shift (Sunday)
      +I;
      T     #H_Out.TotalEvening;  // copy to HMI
ED7:  NOP   0;


NETWORK
TITLE = **** 4.4 - Machine status - Calculated **** Production value Night shift
// Production value Night shift
      A     #Day1;  // Day 1 (Monday)
      JNB   ND1;
      L     #NightDay1Value;  // amount of bodies on day 1 - Night shift (Monday)
      T     #H_Out.TotalNight;  // copy to HMI
ND1:  NOP   0;

      A     #Day2;  // Day 2 (tuesday)
      JNB   ND2;
      L     #NightDay1Value;  // amount of bodies on day 1 - Night shift (Monday)
      L     #NightDay2Value;  // amount of bodies on day 2 - Night shift (Tuesday)
      T     #H_Out.TotalNight;  // copy to HMI
ND2:  NOP   0;

      A     #Day3;  // Day 3 (Wednesday)
      JNB   ND3;
      L     #NightDay1Value;  // amount of bodies on day 1 - Night shift (Monday)
      L     #NightDay2Value;  // amount of bodies on day 2 - Night shift (Tuesday)
      +I;
      L     #NightDay3Value;  // amount of bodies on day 3 - Night shift (Wednesday)
      +I;
      T     #H_Out.TotalNight;  // copy to HMI
ND3:  NOP   0;

      A     #Day4;  // Day 4 (tuesday)
      JNB   ND4;
      L     #NightDay1Value;  // amount of bodies on day 1 - Night shift (Monday)
      L     #NightDay2Value;  // amount of bodies on day 2 - Night shift (Tuesday)
      +I;
      L     #NightDay3Value;  // amount of bodies on day 3 - Night shift (Wednesday)
      +I;
      L     #NightDay4Value;  // amount of bodies on day 4 - Night shift (Thursday)
      +I;
      T     #H_Out.TotalNight;  // copy to HMI
ND4:  NOP   0;

      A     #Day5;  // Day 5 (Friday)
      JNB   ND5;
      L     #NightDay1Value;  // amount of bodies on day 1 - Night shift (Monday)
      L     #NightDay2Value;  // amount of bodies on day 2 - Night shift (Tuesday)
      +I;
      L     #NightDay3Value;  // amount of bodies on day 3 - Night shift (Wednesday)
      +I;
      L     #NightDay4Value;  // amount of bodies on day 4 - Night shift (Thursday)
      +I;
      L     #NightDay5Value;  // amount of bodies on day 5 - Night shift (Friday)
      +I;
      T     #H_Out.TotalNight;  // copy to HMI
ND5:  NOP   0;

      A     #Day6;  // Day 6 (Saturday)
      JNB   ND6;
      L     #NightDay1Value;  // amount of bodies on day 1 - Night shift (Monday)
      L     #NightDay2Value;  // amount of bodies on day 2 - Night shift (Tuesday)
      +I;
      L     #NightDay3Value;  // amount of bodies on day 3 - Night shift (Wednesday)
      +I;
      L     #NightDay4Value;  // amount of bodies on day 4 - Night shift (Thursday)
      +I;
      L     #NightDay5Value;  // amount of bodies on day 5 - Night shift (Friday)
      +I;
      L     #NightDay6Value;  // amount of bodies on day 6 - Night shift (Saturday)
      +I;
      T     #H_Out.TotalNight;  // copy to HMI
ND6:  NOP   0;

      A     #Day7;  // Day 7 (Sunday)
      JNB   ND7;
      L     #NightDay1Value;  // amount of bodies on day 1 - Night shift (Monday)
      L     #NightDay2Value;  // amount of bodies on day 2 - Night shift (Tuesday)
      +I;
      L     #NightDay3Value;  // amount of bodies on day 3 - Night shift (Wednesday)
      +I;
      L     #NightDay4Value;  // amount of bodies on day 4 - Night shift (Thursday)
      +I;
      L     #NightDay5Value;  // amount of bodies on day 5 - Night shift (Friday)
      +I;
      L     #NightDay6Value;  // amount of bodies on day 6 - Night shift (Saturday)
      +I;
      L     #NightDay7Value;  // amount of bodies on day 7 - Evening shift (Sunday)
      +I;
      T     #H_Out.TotalNight;  // copy to HMI
ND7:  NOP   0;


NETWORK
TITLE = **** 4.4 - Machine status - Calculated **** Production value Week on day 1
// Production value Week on day 1
      A     #Day1;  // Day 1 (Monday)
      JNB   day1;
      L     #Day1Value;  // amount of bodies on day 1 (Monday)
      T     #WeekValue;  // copy to HMI
day1: NOP   0;

NETWORK
TITLE = **** 4.4 - Machine status - Calculated **** Production value Week on day 2
// Production value Week on day 2
      A     #Day2;  // Day 2 (tuesday)
      JNB   day2;
      L     #Day1Value;  // amount of bodies on day 1 (Monday)
      L     #Day2Value;  // amount of bodies on day 2 (Tuesday)
      +I;
      T     #WeekValue;  // copy to HMI
day2: NOP   0;

NETWORK
TITLE = **** 4.4 - Machine status - Calculated **** Production value Week on day 3
// Production value Week on day 3
      A     #Day3;  // Day 3 (Wednesday)
      JNB   day3;
      L     #Day1Value;  // amount of bodies on day 1 (Monday)
      L     #Day2Value;  // amount of bodies on day 2 (Tuesday)
      +I;
      L     #Day3Value;  // amount of bodies on day 3 (Wednesday)
      +I;
      T     #WeekValue;  // copy to HMI
day3: NOP   0;

NETWORK
TITLE = **** 4.4 - Machine status - Calculated **** Production value Week on day 4
// Production value Week on day 4
      A     #Day4;  // Day 4 (tuesday)
      JNB   day4;
      L     #Day1Value;  // amount of bodies on day 1 (Monday)
      L     #Day2Value;  // amount of bodies on day 2 (Tuesday)
      +I;
      L     #Day3Value;  // amount of bodies on day 3 (Wednesday)
      +I;
      L     #Day4Value;  // amount of bodies on day 4 (Thursday)
      +I;
      T     #WeekValue;  // copy to HMI
day4: NOP   0;

NETWORK
TITLE = **** 4.4 - Machine status - Calculated **** Production value Week on day 5
// Production value Week on day 5
      A     #Day5;  // Day 5 (Friday)
      JNB   day5;
      L     #Day1Value;  // amount of bodies on day 1 (Monday)
      L     #Day2Value;  // amount of bodies on day 2 (Tuesday)
      +I;
      L     #Day3Value;  // amount of bodies on day 3 (Wednesday)
      +I;
      L     #Day4Value;  // amount of bodies on day 4 (Thursday)
      +I;
      L     #Day5Value;  // amount of bodies on day 5 (Friday)
      +I;
      T     #WeekValue;  // copy to HMI
day5: NOP   0;

NETWORK
TITLE = **** 4.4 - Machine status - Calculated **** Production value Week on day 6
// Production value Week on day 6
      A     #Day6;  // Day 6 (Saturday)
      JNB   day6;
      L     #Day1Value;  // amount of bodies on day 1 (Monday)
      L     #Day2Value;  // amount of bodies on day 2 (Tuesday)
      +I;
      L     #Day3Value;  // amount of bodies on day 3 (Wednesday)
      +I;
      L     #Day4Value;  // amount of bodies on day 4 (Thursday)
      +I;
      L     #Day5Value;  // amount of bodies on day 5 (Friday)
      +I;
      L     #Day6Value;  // amount of bodies on day 6 (Saturday)
      +I;
      T     #WeekValue;  // copy to HMI
day6: NOP   0;

NETWORK
TITLE = **** 4.4 - Machine status - Calculated **** Production value Week on day 7
// Production value Week on day 7
      A     #Day7;  // Day 7 (Sunday)
      JNB   day7;
      L     #Day1Value;  // amount of bodies on day 1 (Monday)
      L     #Day2Value;  // amount of bodies on day 2 (Tuesday)
      +I;
      L     #Day3Value;  // amount of bodies on day 3 (Wednesday)
      +I;
      L     #Day4Value;  // amount of bodies on day 4 (Thursday)
      +I;
      L     #Day5Value;  // amount of bodies on day 5 (Friday)
      +I;
      L     #Day6Value;  // amount of bodies on day 6 (Saturday)
      +I;
      L     #Day7Value;  // amount of bodies on day 7 (Sunday)
      +I;
      T     #WeekValue;  // copy to HMI
day7: NOP   0;

REGION Network 39: **** 4.6 - Machine status - Indications **** Icon Animation
   // Icon Animation for HMI
   IF "TRUE" THEN
       "LSimpleIAnim"(I_SetPos := "FALSE",
                      I_ResetPos := "FALSE",
                      I_Active := "FALSE",
                      I_Invisible := "FALSE",
                      I_OutOfUse := "FALSE",
                      I_AlarmA := "FALSE",
                      I_AlarmB := "FALSE",
                      I_AlarmC := "FALSE",
                      I_AlarmD := "FALSE",
                      I_ManualMode := "FALSE",
                      I_FncSelInHMI := "FALSE",
                      H_IAnim => #H_IAnim);
   END_IF;
END_REGION

REGION Network 40: **** 4.6 - Machine status - Indications **** Animation
   // Animation
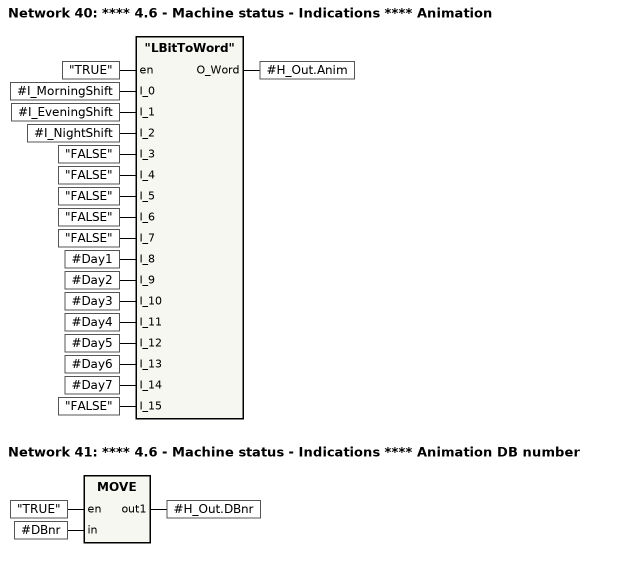
   IF "TRUE" THEN
       "LBitToWord"(I_0 := #I_MorningShift,
                    I_1 := #I_EveningShift,
                    I_2 := #I_NightShift,
                    I_3 := "FALSE",
                    I_4 := "FALSE",
                    I_5 := "FALSE",
                    I_6 := "FALSE",
                    I_7 := "FALSE",
                    I_8 := #Day1,
                    I_9 := #Day2,
                    I_10 := #Day3,
                    I_11 := #Day4,
                    I_12 := #Day5,
                    I_13 := #Day6,
                    I_14 := #Day7,
                    I_15 := "FALSE",
                    O_Word => #H_Out.Anim);
   END_IF;
END_REGION

REGION Network 41: **** 4.6 - Machine status - Indications **** Animation DB number
   // Animation DB number
   IF "TRUE" THEN #H_Out.DBnr := #DBnr; END_IF;
END_REGION

NETWORK
TITLE = **** 8 - Outputs **** Copy of counters for day activities to HMI
// Copy of counters for day activities to HMI
      L     #MorningDay1Value;  // amount of bodies on day 1 - Morning shift (Monday)
      T     #H_Out.MorningDay1Value;  // copy to HMI

      L     #EveningDay1Value;  // amount of bodies on day 1 - Evening shift (Monday)
      T     #H_Out.EveningDay1Value;  // copy to HMI

      L     #NightDay1Value;  // amount of bodies on day 1 - Night shift (Monday)
      T     #H_Out.NightDay1Value;  // copy to HMI

      L     #MorningDay2Value;  // amount of bodies on day 2 - Morning shift (Tuesday)
      T     #H_Out.MorningDay2Value;  // copy to HMI

      L     #EveningDay2Value;  // amount of bodies on day 2 - Evening shift (Tuesday)
      T     #H_Out.EveningDay2Value;  // copy to HMI

      L     #NightDay2Value;  // amount of bodies on day 2 - Night shift (Tuesday)
      T     #H_Out.NightDay2Value;  // copy to HMI

      L     #MorningDay3Value;  // amount of bodies on day 3 - Morning shift (Wednesday)
      T     #H_Out.MorningDay3Value;  // copy to HMI

      L     #EveningDay3Value;  // amount of bodies on day 3 - Evening shift (Wednesday)
      T     #H_Out.EveningDay3Value;  // copy to HMI

      L     #NightDay3Value;  // amount of bodies on day 3 - Night shift (Wednesday)
      T     #H_Out.NightDay3Value;  // copy to HMI

      L     #MorningDay4Value;  // amount of bodies on day 4 - Morning shift (Thursday)
      T     #H_Out.MorningDay4Value;  // copy to HMI

      L     #EveningDay4Value;  // amount of bodies on day 4 - Evening shift (Thursday)
      T     #H_Out.EveningDay4Value;  // copy to HMI

      L     #NightDay4Value;  // amount of bodies on day 4 - Night shift (Thursday)
      T     #H_Out.NightDay4Value;  // copy to HMI

      L     #MorningDay5Value;  // amount of bodies on day 5 - Morning shift (Friday)
      T     #H_Out.MorningDay5Value;  // copy to HMI

      L     #EveningDay5Value;  // amount of bodies on day 5 - Evening shift (Friday)
      T     #H_Out.EveningDay5Value;  // copy to HMI

      L     #NightDay5Value;  // amount of bodies on day 5 - night shift (Friday)
      T     #H_Out.NightDay5Value;  // copy to HMI

      L     #MorningDay6Value;  // amount of bodies on day 6 - Morning shift (Saturday)
      T     #H_Out.MorningDay6Value;  // copy to HMI

      L     #EveningDay6Value;  // amount of bodies on day 6 - Evening shift (Saturday)
      T     #H_Out.EveningDay6Value;  // copy to HMI

      L     #NightDay6Value;  // amount of bodies on day 6 - Night shift (Saturday)
      T     #H_Out.NightDay6Value;  // copy to HMI

      L     #MorningDay7Value;  // amount of bodies on day 7 - Morning shift (Sunday)
      T     #H_Out.MorningDay7Value;  // copy to HMI

      L     #EveningDay7Value;  // amount of bodies on day 7 - Evening shift (Sunday)
      T     #H_Out.EveningDay7Value;  // copy to HMI

      L     #NightDay7Value;  // amount of bodies on day 7 - Night shift (Sunday)
      T     #H_Out.NightDay7Value;  // copy to HMI

NETWORK
TITLE = **** 8 - Outputs **** Copy of counters for summation per day to HMI
// Copy of counters for summation per day to HMI
      L     #Day1Value;  // amount of bodies on day 1 (Monday)
      T     #H_Out.Day1Value;  // copy to HMI

      L     #Day2Value;  // amount of bodies on day 2 (Tuesday)
      T     #H_Out.Day2Value;  // copy to HMI

      L     #Day3Value;  // amount of bodies on day 3 (Wednesday)
      T     #H_Out.Day3Value;  // copy to HMI

      L     #Day4Value;  // amount of bodies on day 4 (Thursday)
      T     #H_Out.Day4Value;  // copy to HMI

      L     #Day5Value;  // amount of bodies on day 5 (Friday)
      T     #H_Out.Day5Value;  // copy to HMI

      L     #Day6Value;  // amount of bodies on day 6 (Saturday)
      T     #H_Out.Day6Value;  // copy to HMI

      L     #Day7Value;  // amount of bodies on day 7 (Sunday)
      T     #H_Out.Day7Value;  // copy to HMI

NETWORK
TITLE = **** 8 - Outputs **** Copy of counter for the complete week to HMI
// Copy of counter for the complete week to HMI
      L     #WeekValue;  // amount of bodies during week
      T     #H_Out.WeekValue;  // copy to HMI

NETWORK
TITLE = **** 8 - Outputs **** Copy of global counter to HMI
// Copy of global counter to HMI
      L     #TotalValue;  // amount of bodies
      T     #H_Out.TotalValue;  // copy to HMI
END_FUNCTION_BLOCK
